% RSLogix 500 project Pump-Protection.RSS, saved by version 8.40.00.08 %
PROJECT "UNTITLED"    % processor: Bul.1763 MicroLogix 1100 Series B %

PROGRAM FILES
  LAD 2   5 rungs
  LAD 3 "I0"  8 rungs
  LAD 4 "CTRL"  5 rungs
  LAD 5 "ALARMS"  7 rungs
  LAD 6 "HOA"  5 rungs

DATA FILES
  O0 OUTPUT  4 elements
  I1 INPUT  6 elements
  S2 STATUS  66 elements
  B3 BINARY  2 elements
  T4 TIMER  4 elements
  C5 COUNTER  1 elements
  R6 CONTROL  1 elements
  N7 INTEGER  3 elements
  F8 FLOAT  1 elements

LADDER 2
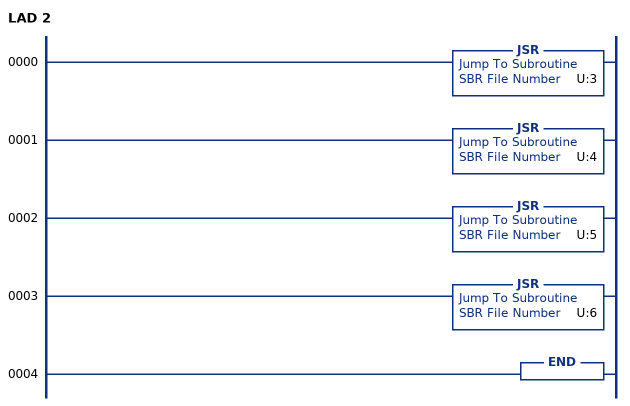
% Rung: 0 %
SOR JSR U:3 EOR
% Rung: 1 %
SOR JSR U:4 EOR
% Rung: 2 %
SOR JSR U:5 EOR
% Rung: 3 %
SOR JSR U:6 EOR
% Rung: 4 %
SOR END EOR

LADDER 3 "I0"
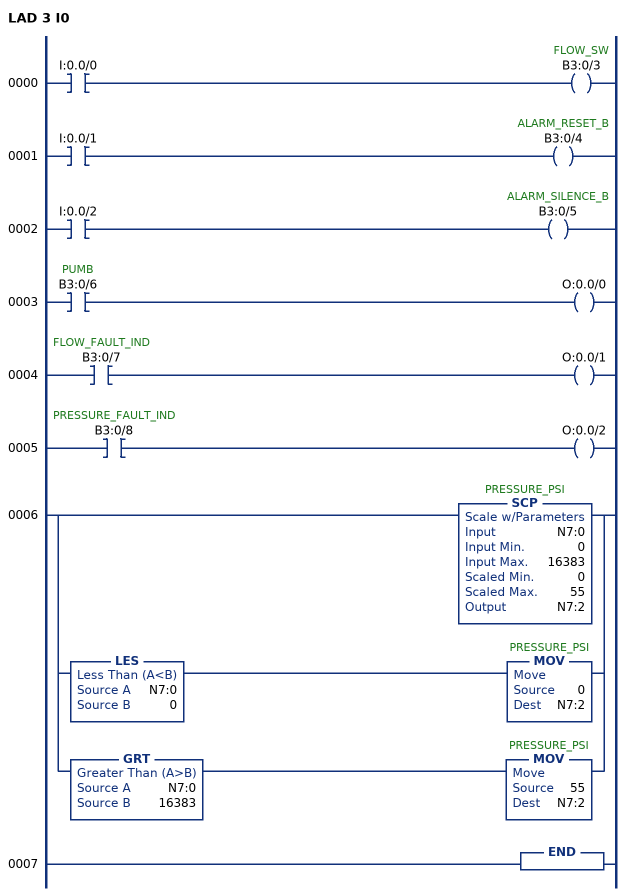
% Rung: 0 %
SOR XIC I:0.0/0 OTE B3:0/3 EOR
%   B3:0/3  FLOW_SW %
% Rung: 1 %
SOR XIC I:0.0/1 OTE B3:0/4 EOR
%   B3:0/4  ALARM_RESET_B %
% Rung: 2 %
SOR XIC I:0.0/2 OTE B3:0/5 EOR
%   B3:0/5  ALARM_SILENCE_B %
% Rung: 3 %
SOR XIC B3:0/6 OTE O:0.0/0 EOR
%   B3:0/6  PUMB %
% Rung: 4 %
SOR XIC B3:0/7 OTE O:0.0/1 EOR
%   B3:0/7  FLOW_FAULT_IND %
% Rung: 5 %
SOR XIC B3:0/8 OTE O:0.0/2 EOR
%   B3:0/8  PRESSURE_FAULT_IND %
% Rung: 6 %
SOR BST SCP N7:0 0 16383 0 55 N7:2 NXB LES N7:0 0 MOV 0 N7:2 NXB GRT N7:0 16383 MOV 55 N7:2 BND EOR
%   N7:2  PRESSURE_PSI %
% Rung: 7 %
SOR END EOR

LADDER 4 "CTRL"
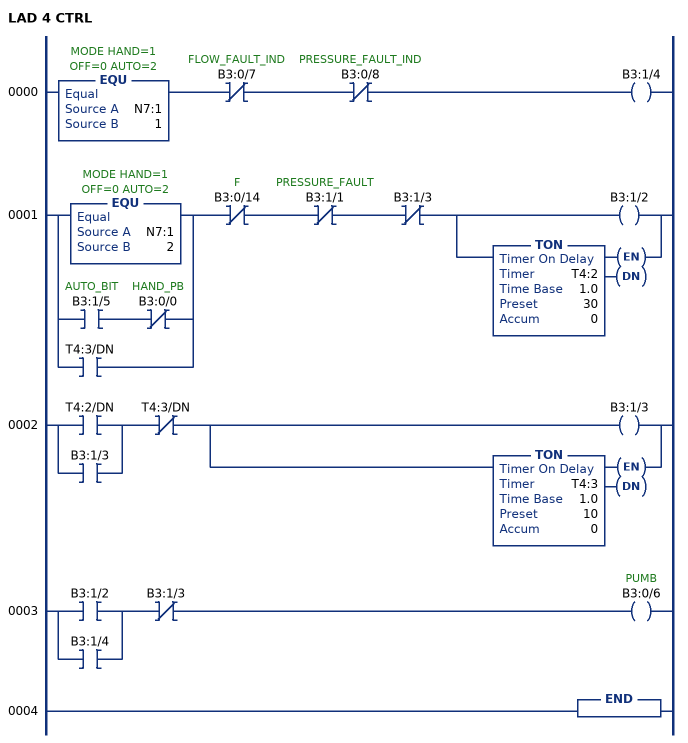
% Rung: 0 %
SOR EQU N7:1 1 XIO B3:0/7 XIO B3:0/8 OTE B3:1/4 EOR
%   N7:1  "MODE HAND=1 OFF=0 AUTO=2" %
%   B3:0/7  FLOW_FAULT_IND %
%   B3:0/8  PRESSURE_FAULT_IND %
% Rung: 1 %
SOR BST BST EQU N7:1 2 NXB XIC B3:1/5 XIO B3:0/0 BND NXB XIC T4:3/DN BND XIO B3:0/14 XIO B3:1/1 XIO B3:1/3 BST OTE B3:1/2 NXB TON T4:2 1.0 30 0 BND EOR
%   N7:1  "MODE HAND=1 OFF=0 AUTO=2" %
%   B3:1/5  AUTO_BIT %
%   B3:0/0  HAND_PB %
%   B3:0/14  F %
%   B3:1/1  PRESSURE_FAULT %
% Rung: 2 %
SOR BST XIC T4:2/DN NXB XIC B3:1/3 BND XIO T4:3/DN BST OTE B3:1/3 NXB TON T4:3 1.0 10 0 BND EOR
% Rung: 3 %
SOR BST XIC B3:1/2 NXB XIC B3:1/4 BND XIO B3:1/3 OTE B3:0/6 EOR
%   B3:0/6  PUMB %
% Rung: 4 %
SOR END EOR

LADDER 5 "ALARMS"
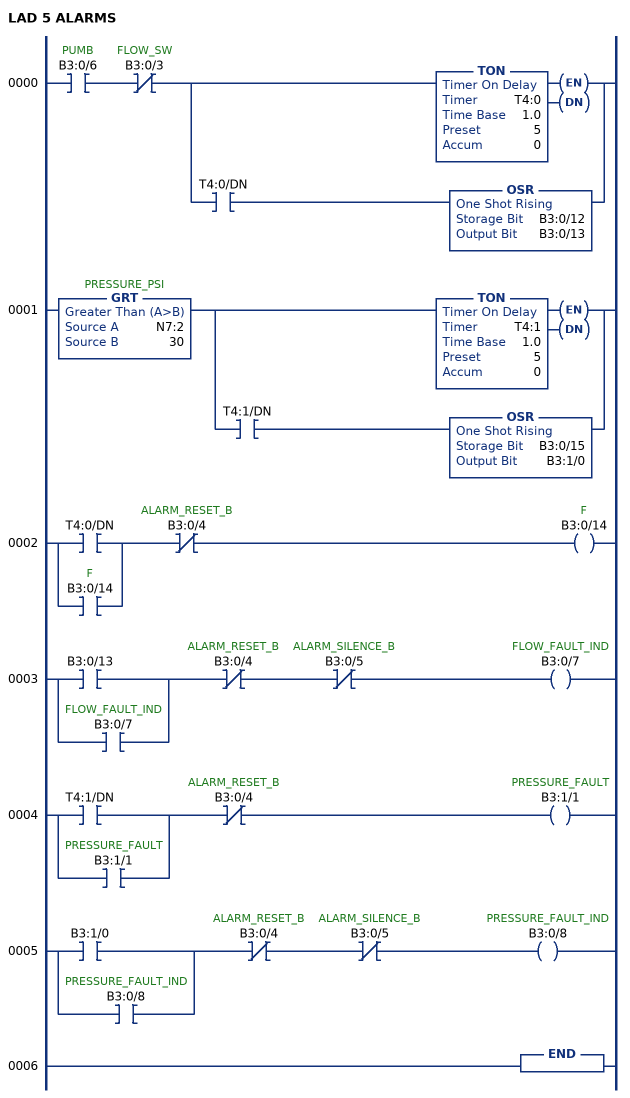
% Rung: 0 %
SOR XIC B3:0/6 XIO B3:0/3 BST TON T4:0 1.0 5 0 NXB XIC T4:0/DN OSR B3:0/12 B3:0/13 BND EOR
%   B3:0/6  PUMB %
%   B3:0/3  FLOW_SW %
% Rung: 1 %
SOR GRT N7:2 30 BST TON T4:1 1.0 5 0 NXB XIC T4:1/DN OSR B3:0/15 B3:1/0 BND EOR
%   N7:2  PRESSURE_PSI %
% Rung: 2 %
SOR BST XIC T4:0/DN NXB XIC B3:0/14 BND XIO B3:0/4 OTE B3:0/14 EOR
%   B3:0/14  F %
%   B3:0/4  ALARM_RESET_B %
% Rung: 3 %
SOR BST XIC B3:0/13 NXB XIC B3:0/7 BND XIO B3:0/4 XIO B3:0/5 OTE B3:0/7 EOR
%   B3:0/7  FLOW_FAULT_IND %
%   B3:0/4  ALARM_RESET_B %
%   B3:0/5  ALARM_SILENCE_B %
% Rung: 4 %
SOR BST XIC T4:1/DN NXB XIC B3:1/1 BND XIO B3:0/4 OTE B3:1/1 EOR
%   B3:1/1  PRESSURE_FAULT %
%   B3:0/4  ALARM_RESET_B %
% Rung: 5 %
SOR BST XIC B3:1/0 NXB XIC B3:0/8 BND XIO B3:0/4 XIO B3:0/5 OTE B3:0/8 EOR
%   B3:0/8  PRESSURE_FAULT_IND %
%   B3:0/4  ALARM_RESET_B %
%   B3:0/5  ALARM_SILENCE_B %
% Rung: 6 %
SOR END EOR

LADDER 6 "HOA"
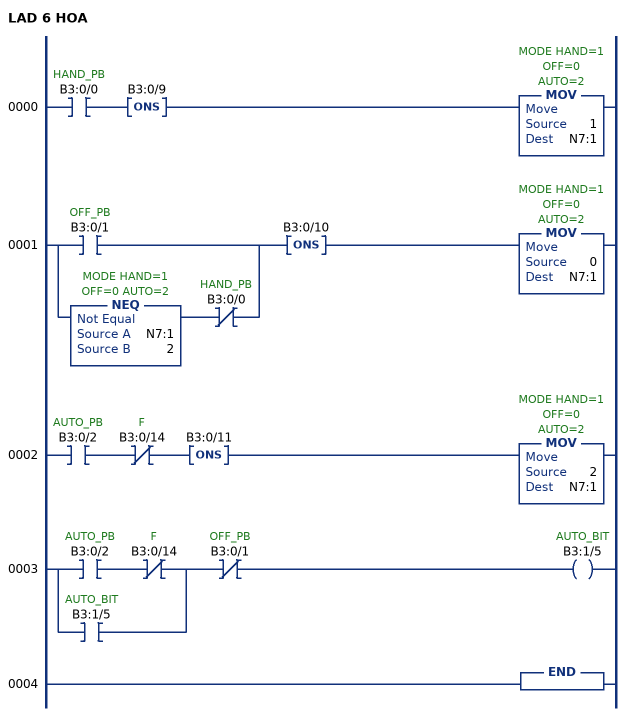
% Rung: 0 %
SOR XIC B3:0/0 ONS B3:0/9 MOV 1 N7:1 EOR
%   B3:0/0  HAND_PB %
%   N7:1  "MODE HAND=1 OFF=0 AUTO=2" %
% Rung: 1 %
SOR BST XIC B3:0/1 NXB NEQ N7:1 2 XIO B3:0/0 BND ONS B3:0/10 MOV 0 N7:1 EOR
%   B3:0/1  OFF_PB %
%   N7:1  "MODE HAND=1 OFF=0 AUTO=2" %
%   B3:0/0  HAND_PB %
% Rung: 2 %
SOR XIC B3:0/2 XIO B3:0/14 ONS B3:0/11 MOV 2 N7:1 EOR
%   B3:0/2  AUTO_PB %
%   B3:0/14  F %
%   N7:1  "MODE HAND=1 OFF=0 AUTO=2" %
% Rung: 3 %
SOR BST XIC B3:0/2 XIO B3:0/14 NXB XIC B3:1/5 BND XIO B3:0/1 OTE B3:1/5 EOR
%   B3:0/2  AUTO_PB %
%   B3:0/14  F %
%   B3:1/5  AUTO_BIT %
%   B3:0/1  OFF_PB %
% Rung: 4 %
SOR END EOR

DATA TABLE (non-zero values as saved)
DATA B3
% B3:0 % 0X4480 0X0020
DATA T4
% .PRE .ACC %
% T4:0 % 5 0
% T4:1 % 5 0
% T4:2 % 30 0
% T4:3 % 10 0
